FUNCTION_BLOCK FB_Busy1
VAR_INPUT
	bSens	 :BOOL;
	tBusy	 :TIME;
	tFree	 :TIME;
	Reset	 :BOOL;
END_VAR
VAR_OUTPUT
	ConvBusy :BOOL := TRUE;
END_VAR
VAR
	Timer1	 :TON;
	Timer2	 :TON;
END_VAR

Timer1 (IN := NOT bSens, PT := tBusy);
IF Timer1.Q THEN ConvBusy := TRUE;
END_IF
Timer2 (IN :=     bSens, PT := tFree);
IF Timer2.Q (*OR Reset*) THEN ConvBusy := FALSE;
END_IF

END_FUNCTION_BLOCK

(* stored: Version 1.1.0.1, ProductVersion 3.1.4024.4
   POU FB_Busy1: Id {2686b548-c476-4a0e-aa14-1d816c51ff17}, SpecialFunc None *)
